{attribute 'qualified_only'}
{attribute 'strict'}
TYPE PrgStates :
(
	START 		:= 0,
	CONNECTING 	:= 1,
	SUBSCRIBING := 2,
	RUN 		:=3
) DINT;
END_TYPE

(* stored: Version 1.1.0.1
   DUT PrgStates: Id {7172dc21-0bf4-0302-36cd-a70aa4380837} *)
